PROGRAM MAIN
VAR
END_VAR

END_PROGRAM

(* stored: Version 1.1.0.1
   POU MAIN: Id {c488fc6a-ca00-41fa-b373-15cd04e6f676} *)
